# EPICS autosave request: ipApp/Db/Rigol_DG4000_settings.req
$(P)$(R)UserWaveform
$(P)$(R)UserWf1Size
$(P)$(R)UserWf2Size
$(P)$(R)UserWf3Size
$(P)$(R)UserWf4Size
